% RSLogix 500 project CCHDUMP_BAK004.RSS, saved by version 11.00.00.00 %
PROJECT "CCHDUMP"    % processor: MicroLogix 1400 %

PROGRAM FILES
  LAD 2   44 rungs

DATA FILES
  O0 OUTPUT  6 elements
  I1 INPUT  8 elements
  S2 STATUS  66 elements
  B3 BINARY  3 elements
  T4 TIMER  19 elements
  C5 COUNTER  1 elements
  R6 CONTROL  1 elements
  N7 INTEGER  1 elements
  F8 FLOAT  1 elements

LADDER 2
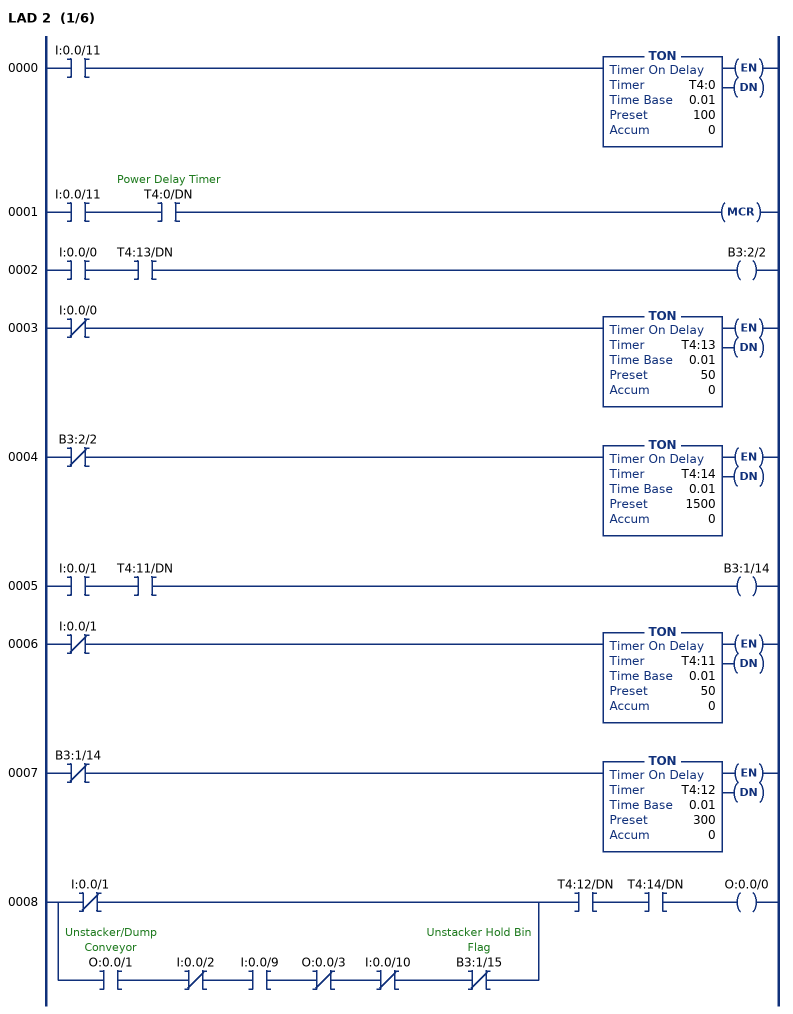
% Rung: 0 %
SOR XIC I:0.0/11 TON T4:0 0.01 100 0 EOR
% Rung: 1 %
SOR XIC I:0.0/11 XIC T4:0/DN MCR EOR
%   T4:0/DN  "Power Delay Timer" %
% Rung: 2 %
SOR XIC I:0.0/0 XIC T4:13/DN OTE B3:2/2 EOR
% Rung: 3 %
SOR XIO I:0.0/0 TON T4:13 0.01 50 0 EOR
% Rung: 4 %
SOR XIO B3:2/2 TON T4:14 0.01 1500 0 EOR
% Rung: 5 %
SOR XIC I:0.0/1 XIC T4:11/DN OTE B3:1/14 EOR
% Rung: 6 %
SOR XIO I:0.0/1 TON T4:11 0.01 50 0 EOR
% Rung: 7 %
SOR XIO B3:1/14 TON T4:12 0.01 300 0 EOR
% Rung: 8 %
SOR BST XIO I:0.0/1 NXB XIC O:0.0/1 XIO I:0.0/2 XIC I:0.0/9 XIO O:0.0/3 XIO I:0.0/10 XIO B3:1/15 BND XIC T4:12/DN XIC T4:14/DN OTE O:0.0/0 EOR
%   O:0.0/1  "Unstacker/Dump Conveyor" %
%   B3:1/15  "Unstacker Hold Bin Flag" %

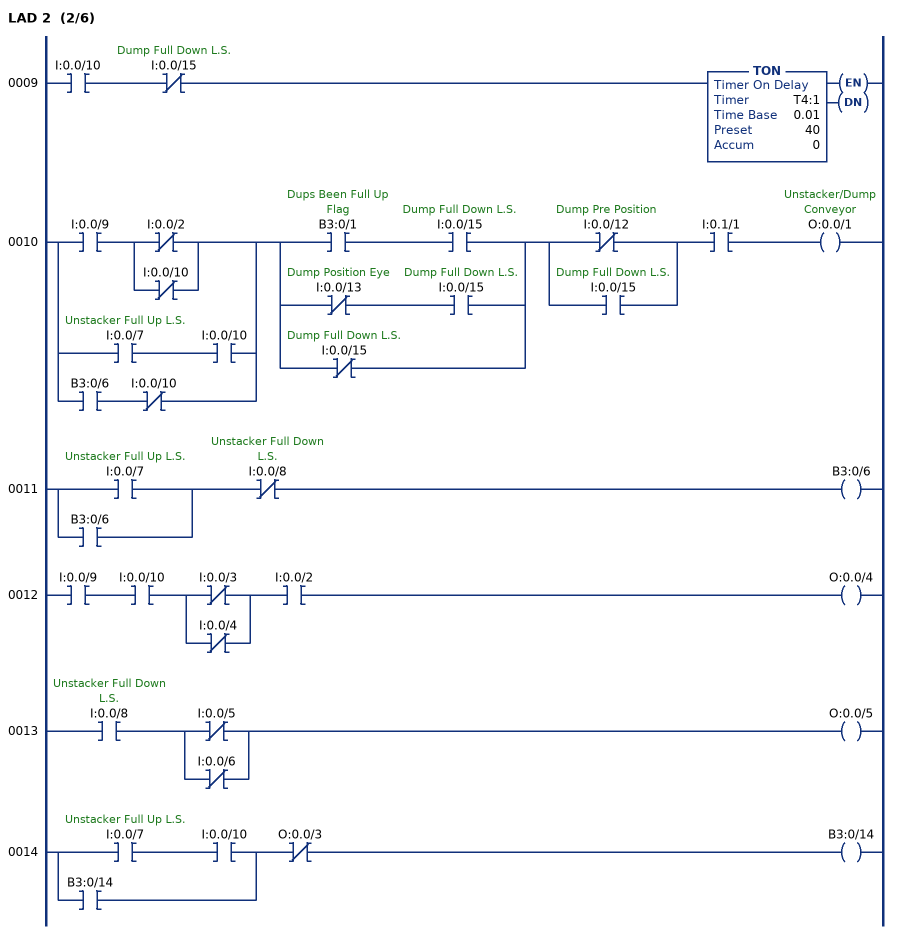
% Rung: 9 %
SOR XIC I:0.0/10 XIO I:0.0/15 TON T4:1 0.01 40 0 EOR
%   I:0.0/15  "Dump Full Down L.S." %
% Rung: 10 %
SOR BST XIC I:0.0/9 BST XIO I:0.0/2 NXB XIO I:0.0/10 BND NXB XIC I:0.0/7 XIC I:0.0/10 NXB XIC B3:0/6 XIO I:0.0/10 BND BST XIC B3:0/1 XIC I:0.0/15 NXB XIO I:0.0/13 XIC I:0.0/15 NXB XIO I:0.0/15 BND BST XIO I:0.0/12 NXB XIC I:0.0/15 BND XIC I:0.1/1 OTE O:0.0/1 EOR
%   I:0.0/7  "Unstacker Full Up L.S." %
%   B3:0/1  "Dups Been Full Up Flag" %
%   I:0.0/15  "Dump Full Down L.S." %
%   I:0.0/13  "Dump Position Eye" %
%   I:0.0/12  "Dump Pre Position" %
%   O:0.0/1  "Unstacker/Dump Conveyor" %
% Rung: 11 %
SOR BST XIC I:0.0/7 NXB XIC B3:0/6 BND XIO I:0.0/8 OTE B3:0/6 EOR
%   I:0.0/7  "Unstacker Full Up L.S." %
%   I:0.0/8  "Unstacker Full Down L.S." %
% Rung: 12 %
SOR XIC I:0.0/9 XIC I:0.0/10 BST XIO I:0.0/3 NXB XIO I:0.0/4 BND XIC I:0.0/2 OTE O:0.0/4 EOR
% Rung: 13 %
SOR XIC I:0.0/8 BST XIO I:0.0/5 NXB XIO I:0.0/6 BND OTE O:0.0/5 EOR
%   I:0.0/8  "Unstacker Full Down L.S." %
% Rung: 14 %
SOR BST XIC I:0.0/7 XIC I:0.0/10 NXB XIC B3:0/14 BND XIO O:0.0/3 OTE B3:0/14 EOR
%   I:0.0/7  "Unstacker Full Up L.S." %

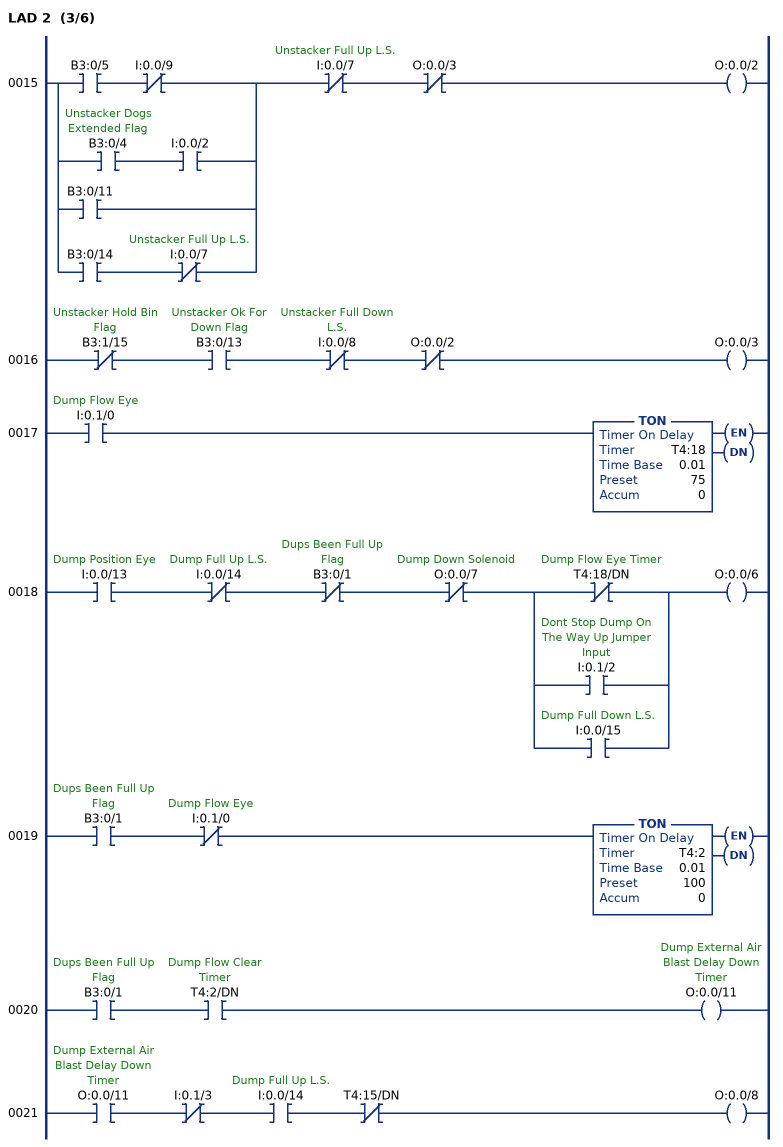
% Rung: 15 %
SOR BST XIC B3:0/5 XIO I:0.0/9 NXB XIC B3:0/4 XIC I:0.0/2 NXB XIC B3:0/11 NXB XIC B3:0/14 XIO I:0.0/7 BND XIO I:0.0/7 XIO O:0.0/3 OTE O:0.0/2 EOR
%   B3:0/4  "Unstacker Dogs Extended Flag" %
%   I:0.0/7  "Unstacker Full Up L.S." %
% Rung: 16 %
SOR XIO B3:1/15 XIC B3:0/13 XIO I:0.0/8 XIO O:0.0/2 OTE O:0.0/3 EOR
%   B3:1/15  "Unstacker Hold Bin Flag" %
%   B3:0/13  "Unstacker Ok For Down Flag" %
%   I:0.0/8  "Unstacker Full Down L.S." %
% Rung: 17 %
SOR XIC I:0.1/0 TON T4:18 0.01 75 0 EOR
%   I:0.1/0  "Dump Flow Eye" %
% Rung: 18 %
SOR XIC I:0.0/13 XIO I:0.0/14 XIO B3:0/1 XIO O:0.0/7 BST XIO T4:18/DN NXB XIC I:0.1/2 NXB XIC I:0.0/15 BND OTE O:0.0/6 EOR
%   I:0.0/13  "Dump Position Eye" %
%   I:0.0/14  "Dump Full Up L.S." %
%   B3:0/1  "Dups Been Full Up Flag" %
%   O:0.0/7  "Dump Down Solenoid" %
%   T4:18/DN  "Dump Flow Eye Timer" %
%   I:0.1/2  "Dont Stop Dump On The Way Up Jumper Input" %
%   I:0.0/15  "Dump Full Down L.S." %
% Rung: 19 %
SOR XIC B3:0/1 XIO I:0.1/0 TON T4:2 0.01 100 0 EOR
%   B3:0/1  "Dups Been Full Up Flag" %
%   I:0.1/0  "Dump Flow Eye" %
% Rung: 20 %
SOR XIC B3:0/1 XIC T4:2/DN OTE O:0.0/11 EOR
%   B3:0/1  "Dups Been Full Up Flag" %
%   T4:2/DN  "Dump Flow Clear Timer" %
%   O:0.0/11  "Dump External Air Blast Delay Down Timer" %
% Rung: 21 %
SOR XIC O:0.0/11 XIO I:0.1/3 XIC I:0.0/14 XIO T4:15/DN OTE O:0.0/8 EOR
%   O:0.0/11  "Dump External Air Blast Delay Down Timer" %
%   I:0.0/14  "Dump Full Up L.S." %

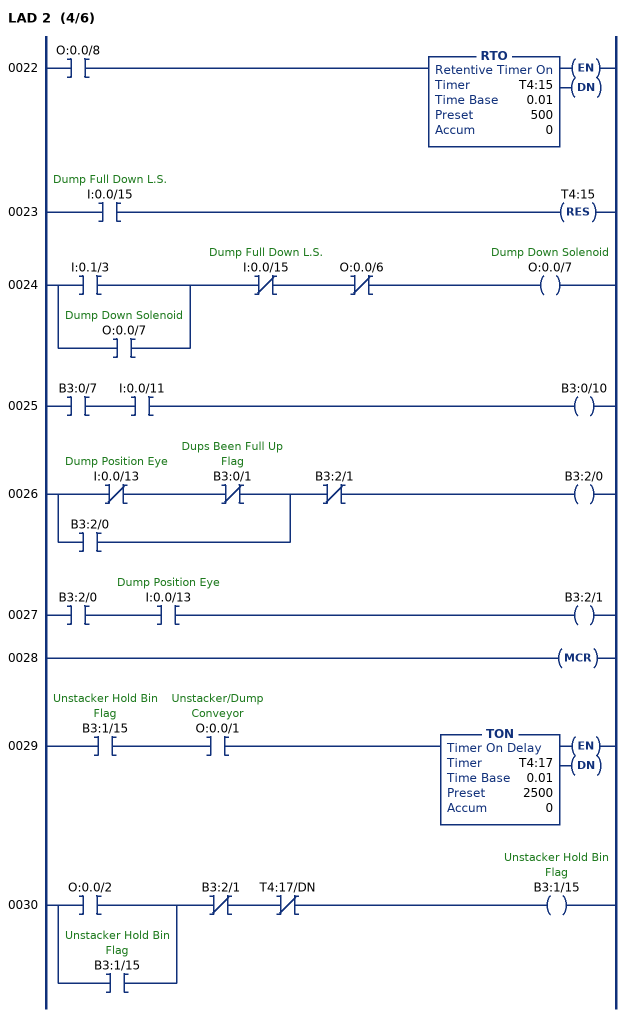
% Rung: 22 %
SOR XIC O:0.0/8 RTO T4:15 0.01 500 0 EOR
% Rung: 23 %
SOR XIC I:0.0/15 RES T4:15 EOR
%   I:0.0/15  "Dump Full Down L.S." %
% Rung: 24 %
SOR BST XIC I:0.1/3 NXB XIC O:0.0/7 BND XIO I:0.0/15 XIO O:0.0/6 OTE O:0.0/7 EOR
%   O:0.0/7  "Dump Down Solenoid" %
%   I:0.0/15  "Dump Full Down L.S." %
% Rung: 25 %
SOR XIC B3:0/7 XIC I:0.0/11 OTE B3:0/10 EOR
% Rung: 26 %
SOR BST XIO I:0.0/13 XIO B3:0/1 NXB XIC B3:2/0 BND XIO B3:2/1 OTE B3:2/0 EOR
%   I:0.0/13  "Dump Position Eye" %
%   B3:0/1  "Dups Been Full Up Flag" %
% Rung: 27 %
SOR XIC B3:2/0 XIC I:0.0/13 OTE B3:2/1 EOR
%   I:0.0/13  "Dump Position Eye" %
% Rung: 28 %
SOR MCR EOR
% Rung: 29 %
SOR XIC B3:1/15 XIC O:0.0/1 TON T4:17 0.01 2500 0 EOR
%   B3:1/15  "Unstacker Hold Bin Flag" %
%   O:0.0/1  "Unstacker/Dump Conveyor" %
% Rung: 30 %
SOR BST XIC O:0.0/2 NXB XIC B3:1/15 BND XIO B3:2/1 XIO T4:17/DN OTE B3:1/15 EOR
%   B3:1/15  "Unstacker Hold Bin Flag" %

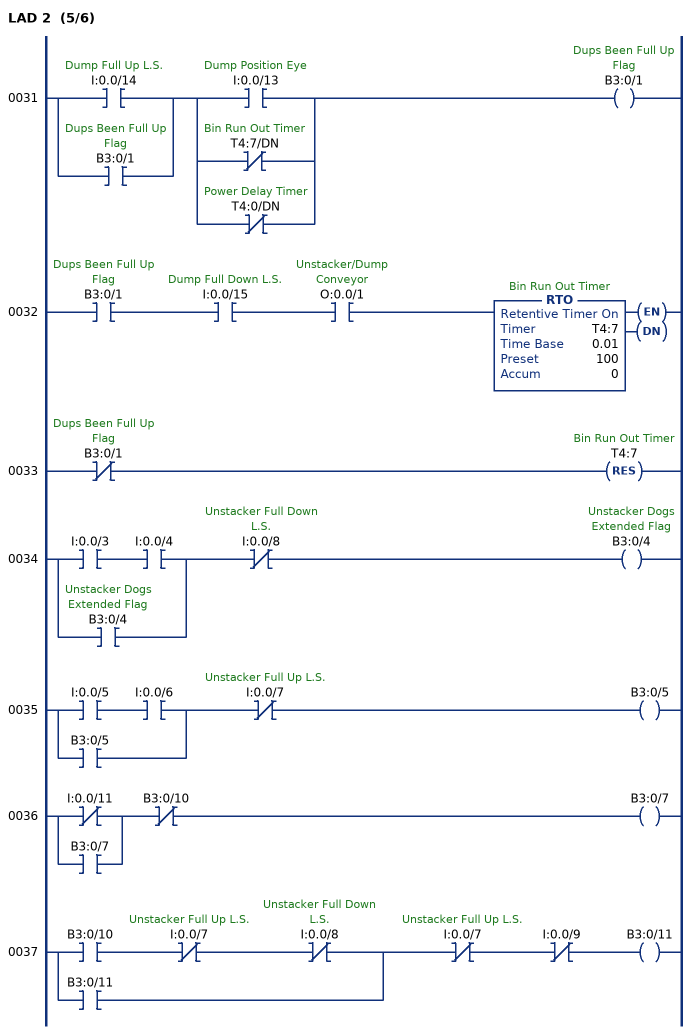
% Rung: 31 %
SOR BST XIC I:0.0/14 NXB XIC B3:0/1 BND BST XIC I:0.0/13 NXB XIO T4:7/DN NXB XIO T4:0/DN BND OTE B3:0/1 EOR
%   I:0.0/14  "Dump Full Up L.S." %
%   B3:0/1  "Dups Been Full Up Flag" %
%   I:0.0/13  "Dump Position Eye" %
%   T4:7/DN  "Bin Run Out Timer" %
%   T4:0/DN  "Power Delay Timer" %
% Rung: 32 %
SOR XIC B3:0/1 XIC I:0.0/15 XIC O:0.0/1 RTO T4:7 0.01 100 0 EOR
%   B3:0/1  "Dups Been Full Up Flag" %
%   I:0.0/15  "Dump Full Down L.S." %
%   O:0.0/1  "Unstacker/Dump Conveyor" %
%   T4:7  "Bin Run Out Timer" %
% Rung: 33 %
SOR XIO B3:0/1 RES T4:7 EOR
%   B3:0/1  "Dups Been Full Up Flag" %
%   T4:7  "Bin Run Out Timer" %
% Rung: 34 %
SOR BST XIC I:0.0/3 XIC I:0.0/4 NXB XIC B3:0/4 BND XIO I:0.0/8 OTE B3:0/4 EOR
%   B3:0/4  "Unstacker Dogs Extended Flag" %
%   I:0.0/8  "Unstacker Full Down L.S." %
% Rung: 35 %
SOR BST XIC I:0.0/5 XIC I:0.0/6 NXB XIC B3:0/5 BND XIO I:0.0/7 OTE B3:0/5 EOR
%   I:0.0/7  "Unstacker Full Up L.S." %
% Rung: 36 %
SOR BST XIO I:0.0/11 NXB XIC B3:0/7 BND XIO B3:0/10 OTE B3:0/7 EOR
% Rung: 37 %
SOR BST XIC B3:0/10 XIO I:0.0/7 XIO I:0.0/8 NXB XIC B3:0/11 BND XIO I:0.0/7 XIO I:0.0/9 OTE B3:0/11 EOR
%   I:0.0/7  "Unstacker Full Up L.S." %
%   I:0.0/8  "Unstacker Full Down L.S." %

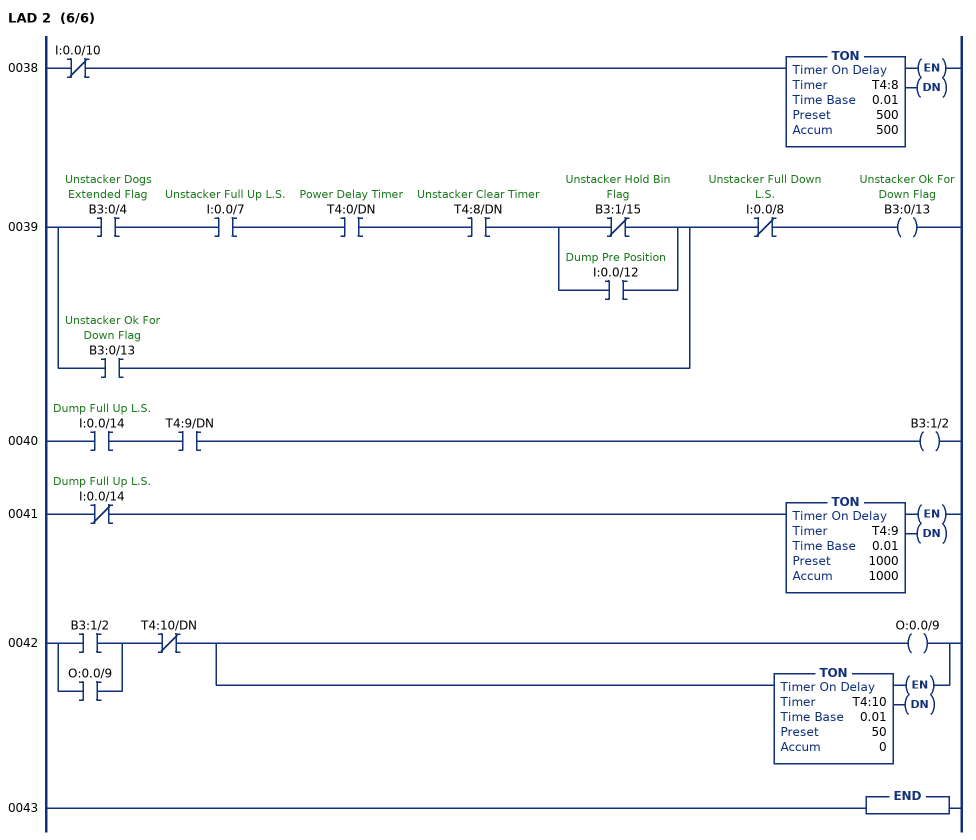
% Rung: 38 %
SOR XIO I:0.0/10 TON T4:8 0.01 500 500 EOR
% Rung: 39 %
SOR BST XIC B3:0/4 XIC I:0.0/7 XIC T4:0/DN XIC T4:8/DN BST XIO B3:1/15 NXB XIC I:0.0/12 BND NXB XIC B3:0/13 BND XIO I:0.0/8 OTE B3:0/13 EOR
%   B3:0/4  "Unstacker Dogs Extended Flag" %
%   I:0.0/7  "Unstacker Full Up L.S." %
%   T4:0/DN  "Power Delay Timer" %
%   T4:8/DN  "Unstacker Clear Timer" %
%   B3:1/15  "Unstacker Hold Bin Flag" %
%   I:0.0/12  "Dump Pre Position" %
%   B3:0/13  "Unstacker Ok For Down Flag" %
%   I:0.0/8  "Unstacker Full Down L.S." %
% Rung: 40 %
SOR XIC I:0.0/14 XIC T4:9/DN OTE B3:1/2 EOR
%   I:0.0/14  "Dump Full Up L.S." %
% Rung: 41 %
SOR XIO I:0.0/14 TON T4:9 0.01 1000 1000 EOR
%   I:0.0/14  "Dump Full Up L.S." %
% Rung: 42 %
SOR BST XIC B3:1/2 NXB XIC O:0.0/9 BND XIO T4:10/DN BST OTE O:0.0/9 NXB TON T4:10 0.01 50 0 BND EOR
% Rung: 43 %
SOR END EOR

REVISION NOTES
  0: Eidenburg Bin Dump

DATA TABLE (non-zero values as saved)
DATA B3
% B3:0 % 0X00A2 0X0000 0X0000
DATA T4
% .PRE .ACC %
% T4:0 % 100 0
% T4:1 % 40 0
% T4:2 % 100 0
% T4:3 % 100 0
% T4:4 % 50 0
% T4:5 % 100 0
% T4:6 % 50 0
% T4:7 % 100 0
% T4:8 % 500 500
% T4:9 % 1000 1000
% T4:10 % 50 0
% T4:11 % 50 0
% T4:12 % 300 0
% T4:13 % 50 0
% T4:14 % 1500 0
% T4:15 % 500 0
% T4:16 % 100 0
% T4:17 % 2500 0
% T4:18 % 75 0
